ABB RobotStudio station: robotstudio-pick-place.rsstn

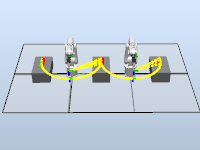
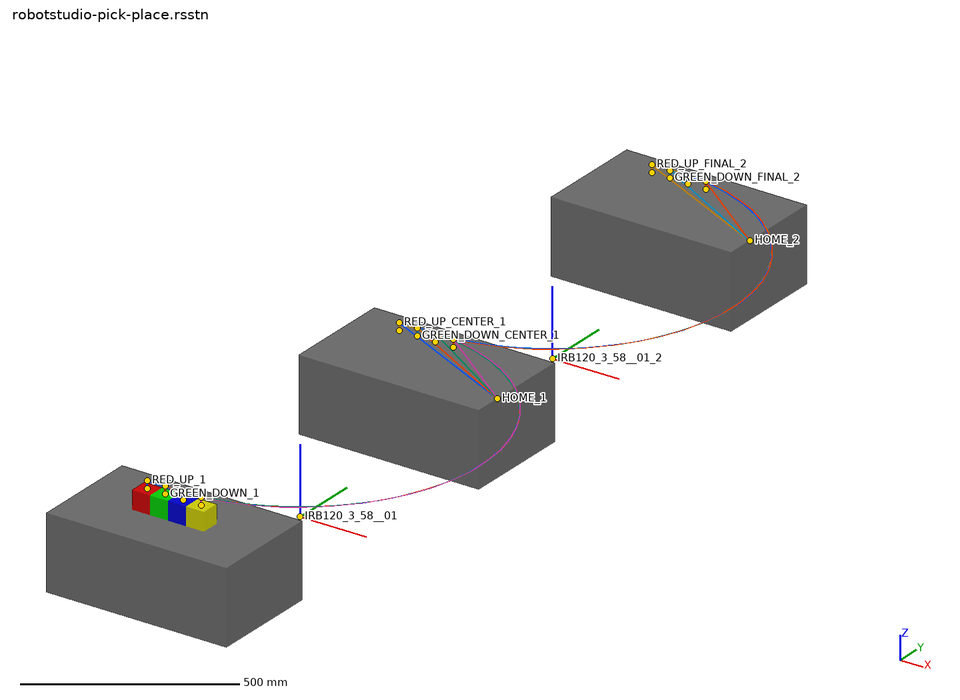
[picture v1: parts stored in the station drawn from their meshes, with robot base, taught points and paths (robot models come from the ABB library and are not in the file)]
Station robotstudio-pick-place (saved by RobotStudio 21.3.9648.0)
Controller PickPlace
  mechanical unit ROB_1: IRB120_3_58__01, 6 joints, base frame (0, 0, 0) mm
  mechanical unit ROB_2: IRB120_3_58__01_2, 6 joints, base frame (0, 1000, 0) mm
Layout (positions relative to the parent item):
  - IRB120_3_58__01 [mechanism, from Robots\IRB120_3_58_G_01.rslib] at (0, 0, 0) mm; joint values [0, 0, 0, 0, 0.5236, 0] (rad or m)
  - IRB120_3_58__01_2 [mechanism, from Robots\IRB120_3_58_G_01.rslib] at (0, 1000, 0) mm; joint values [0, 0, 0, 0, 0.5236, 0] (rad or m)
  - MyTool [mechanism, from Training Objects\myTool.rslib] at (364.35, 0, 594) mm, rotated rx 180 ry 60 rz 180 deg
  - CUBE_1 [part] at (-100, 0, -50) mm, size 50 x 50 x 50 mm
  - CUBE_2 [part] at (-50, 0, -50) mm, size 50 x 50 x 50 mm
  - CUBE_3 [part] at (0, 0, -50) mm, size 50 x 50 x 50 mm
  - CUBE_4 [part] at (50, 0, -50) mm, size 50 x 50 x 50 mm
  - CUBE_1_CENTER [part] at (-100, 1000, -50) mm, size 50 x 50 x 50 mm
  - CUBE_2_CENTER [part] at (-50, 1000, -50) mm, size 50 x 50 x 50 mm
  - CUBE_3_CENTER [part] at (0, 1000, -50) mm, size 50 x 50 x 50 mm
  - CUBE_4_CENTER [part] at (50, 1000, -50) mm, size 50 x 50 x 50 mm
  - CUBE_1_FINAL [part] at (-100, 2000, -50) mm, size 50 x 50 x 50 mm
  - CUBE_2_FINAL [part] at (-50, 2000, -50) mm, size 50 x 50 x 50 mm
  - CUBE_3_FINAL [part] at (0, 2000, -50) mm, size 50 x 50 x 50 mm
  - CUBE_4_FINAL [part] at (50, 2000, -50) mm, size 50 x 50 x 50 mm
  - TABLE_1 [part], size 500 x 300 x 200 mm
  - TABLE_2 [part] at (0, 1000, 0) mm, size 500 x 300 x 200 mm
  - TABLE_3 [part] at (0, 2000, 0) mm, size 500 x 300 x 200 mm
  - MyTool_2 [mechanism, from Training Objects\myTool.rslib] at (364.35, 1000, 594) mm, rotated rx 180 ry 60 rz 180 deg
  - Positioner [smart component, from Components\Positioner.rslib]
      properties: Object=CUBE_1; Position=[0 0 0]; Orientation=[0 0 0]; Reference=Global; ReferenceObject=(none)
  - CollisionSensor [smart component, from Components\CollisionSensor.rslib]
      properties: Object1=MyTool; Object2=CUBE_1; NearMiss=0.01; Part1=(none); Part2=(none); CollisionType=0
  - CollisionSensor_2 [smart component, from Components\CollisionSensor.rslib]
      properties: Object1=MyTool; Object2=CUBE_1_CENTER; NearMiss=0.01; Part1=(none); Part2=(none); CollisionType=0
  - Attacher [smart component, from Components\Attacher.rslib]
      properties: Parent=MyTool; Flange=0; Child=CUBE_1; Mount=false; Offset=[0 0 0]; Orientation=[0 0 0]
  - Detacher [smart component, from Components\Detacher.rslib]
      properties: Child=CUBE_1; KeepPosition=true
  - Positioner_2 [smart component, from Components\Positioner.rslib]
      properties: Object=CUBE_1_CENTER; Position=[0 0 0]; Orientation=[0 0 0]; Reference=Global; ReferenceObject=(none)
  - CollisionSensor_3 [smart component, from Components\CollisionSensor.rslib]
      properties: Object1=MyTool_2; Object2=CUBE_1_CENTER; NearMiss=0.01; Part1=(none); Part2=(none); CollisionType=0
  - CollisionSensor_4 [smart component, from Components\CollisionSensor.rslib]
      properties: Object1=MyTool_2; Object2=CUBE_1_FINAL; NearMiss=0.01; Part1=(none); Part2=(none); CollisionType=0
  - Attacher_2 [smart component, from Components\Attacher.rslib]
      properties: Parent=MyTool_2; Flange=0; Child=CUBE_1; Mount=false; Offset=[0 0 0]; Orientation=[0 0 0]
  - Detacher_2 [smart component, from Components\Detacher.rslib]
      properties: Child=CUBE_1; KeepPosition=true
  - Positioner_3 [smart component, from Components\Positioner.rslib]
      properties: Object=(none); Position=[0 0 0]; Orientation=[0 0 0]; Reference=Global; ReferenceObject=(none)
  - CollisionSensor_5 [smart component, from Components\CollisionSensor.rslib]
      properties: Object1=MyTool; Object2=CUBE_2; NearMiss=0.01; Part1=(none); Part2=(none); CollisionType=0
  - CollisionSensor_6 [smart component, from Components\CollisionSensor.rslib]
      properties: Object1=MyTool; Object2=CUBE_2_CENTER; NearMiss=0.01; Part1=(none); Part2=(none); CollisionType=0
  - Attacher_3 [smart component, from Components\Attacher.rslib]
      properties: Parent=MyTool; Flange=0; Child=CUBE_2; Mount=false; Offset=[0 0 0]; Orientation=[0 0 0]
  - Detacher_3 [smart component, from Components\Detacher.rslib]
      properties: Child=CUBE_2; KeepPosition=true
  - Positioner_4 [smart component, from Components\Positioner.rslib]
      properties: Object=(none); Position=[0 0 0]; Orientation=[0 0 0]; Reference=Global; ReferenceObject=(none)
  - CollisionSensor_7 [smart component, from Components\CollisionSensor.rslib]
      properties: Object1=MyTool_2; Object2=CUBE_2_CENTER; NearMiss=0.01; Part1=(none); Part2=(none); CollisionType=0
  - CollisionSensor_8 [smart component, from Components\CollisionSensor.rslib]
      properties: Object1=MyTool_2; Object2=CUBE_2_FINAL; NearMiss=0.01; Part1=(none); Part2=(none); CollisionType=0
  - Attacher_4 [smart component, from Components\Attacher.rslib]
      properties: Parent=MyTool_2; Flange=0; Child=CUBE_2; Mount=false; Offset=[0 0 0]; Orientation=[0 0 0]
  - Detacher_4 [smart component, from Components\Detacher.rslib]
      properties: Child=CUBE_2; KeepPosition=true
  - Positioner_5 [smart component, from Components\Positioner.rslib]
      properties: Object=(none); Position=[0 0 0]; Orientation=[0 0 0]; Reference=Global; ReferenceObject=(none)
  - CollisionSensor_9 [smart component, from Components\CollisionSensor.rslib]
      properties: Object1=MyTool; Object2=CUBE_3; NearMiss=0.01; Part1=(none); Part2=(none); CollisionType=0
  - CollisionSensor_10 [smart component, from Components\CollisionSensor.rslib]
      properties: Object1=MyTool; Object2=CUBE_3_CENTER; NearMiss=0.01; Part1=(none); Part2=(none); CollisionType=0
  - Attacher_5 [smart component, from Components\Attacher.rslib]
      properties: Parent=MyTool; Flange=0; Child=CUBE_3; Mount=false; Offset=[0 0 0]; Orientation=[0 0 0]
  - Detacher_5 [smart component, from Components\Detacher.rslib]
      properties: Child=CUBE_3; KeepPosition=true
  - Positioner_6 [smart component, from Components\Positioner.rslib]
      properties: Object=(none); Position=[0 0 0]; Orientation=[0 0 0]; Reference=Global; ReferenceObject=(none)
  - CollisionSensor_11 [smart component, from Components\CollisionSensor.rslib]
      properties: Object1=MyTool_2; Object2=CUBE_3; NearMiss=0.01; Part1=(none); Part2=(none); CollisionType=0
  - CollisionSensor_12 [smart component, from Components\CollisionSensor.rslib]
      properties: Object1=MyTool_2; Object2=CUBE_3_FINAL; NearMiss=0.01; Part1=(none); Part2=(none); CollisionType=0
  - Attacher_6 [smart component, from Components\Attacher.rslib]
      properties: Parent=MyTool_2; Flange=0; Child=CUBE_3; Mount=false; Offset=[0 0 0]; Orientation=[0 0 0]
  - Detacher_6 [smart component, from Components\Detacher.rslib]
      properties: Child=CUBE_3; KeepPosition=true
  - Positioner_7 [smart component, from Components\Positioner.rslib]
      properties: Object=(none); Position=[0 0 0]; Orientation=[0 0 0]; Reference=Global; ReferenceObject=(none)
  - CollisionSensor_13 [smart component, from Components\CollisionSensor.rslib]
      properties: Object1=MyTool; Object2=CUBE_4; NearMiss=0.01; Part1=(none); Part2=(none); CollisionType=0
  - CollisionSensor_14 [smart component, from Components\CollisionSensor.rslib]
      properties: Object1=MyTool; Object2=CUBE_4_CENTER; NearMiss=0.01; Part1=(none); Part2=(none); CollisionType=0
  - Attacher_7 [smart component, from Components\Attacher.rslib]
      properties: Parent=MyTool; Flange=0; Child=CUBE_4; Mount=false; Offset=[0 0 0]; Orientation=[0 0 0]
  - Detacher_7 [smart component, from Components\Detacher.rslib]
      properties: Child=CUBE_4; KeepPosition=true
  - Positioner_8 [smart component, from Components\Positioner.rslib]
      properties: Object=CUBE_4_CENTER; Position=[0 0 0]; Orientation=[0 0 0]; Reference=Global; ReferenceObject=(none)
  - CollisionSensor_15 [smart component, from Components\CollisionSensor.rslib]
      properties: Object1=MyTool_2; Object2=CUBE_4_CENTER; NearMiss=0.01; Part1=(none); Part2=(none); CollisionType=0
  - CollisionSensor_16 [smart component, from Components\CollisionSensor.rslib]
      properties: Object1=MyTool_2; Object2=CUBE_4_FINAL; NearMiss=0.01; Part1=(none); Part2=(none); CollisionType=0
  - Attacher_8 [smart component, from Components\Attacher.rslib]
      properties: Parent=MyTool_2; Flange=0; Child=CUBE_4; Mount=false; Offset=[0 0 0]; Orientation=[0 0 0]
  - Detacher_8 [smart component, from Components\Detacher.rslib]
      properties: Child=CUBE_4; KeepPosition=true
Attachment: MyTool is attached to IRB120_3_58__01 / Link6
Attachment: MyTool_2 is attached to IRB120_3_58__01_2 / Link6
Station signals: DI Digital1, DI Digital2, DI Digital3, DI Digital4, DI Digital5, DI Digital6, DI Digital7, DI Digital8
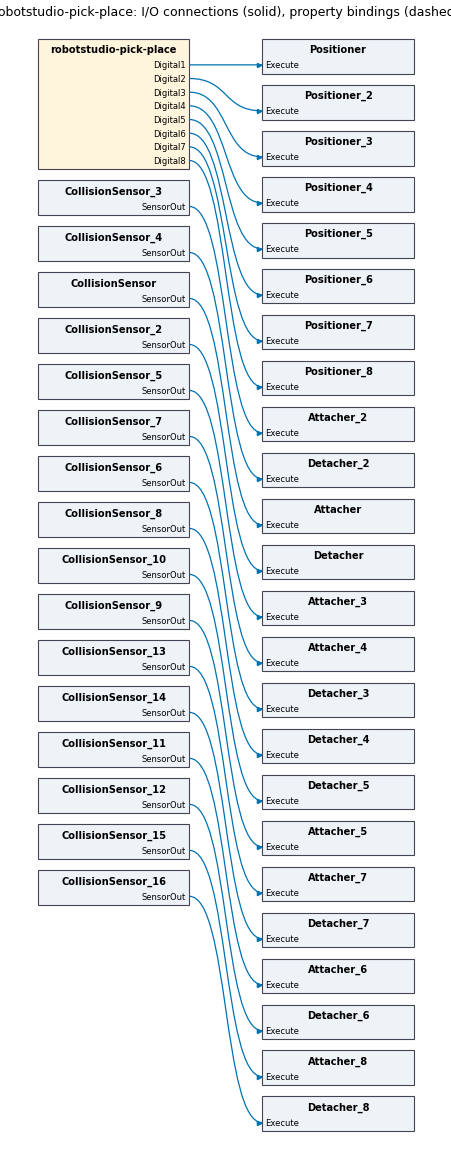
Station logic (signal -> signal, property => property):
  robotstudio-pick-place.Digital1 -> Positioner.Execute
  robotstudio-pick-place.Digital2 -> Positioner_2.Execute
  CollisionSensor_3.SensorOut -> Attacher_2.Execute
  CollisionSensor_4.SensorOut -> Detacher_2.Execute
  CollisionSensor.SensorOut -> Attacher.Execute
  CollisionSensor_2.SensorOut -> Detacher.Execute
  robotstudio-pick-place.Digital3 -> Positioner_3.Execute
  robotstudio-pick-place.Digital4 -> Positioner_4.Execute
  CollisionSensor_5.SensorOut -> Attacher_3.Execute
  CollisionSensor_7.SensorOut -> Attacher_4.Execute
  CollisionSensor_6.SensorOut -> Detacher_3.Execute
  CollisionSensor_8.SensorOut -> Detacher_4.Execute
  robotstudio-pick-place.Digital5 -> Positioner_5.Execute
  CollisionSensor_10.SensorOut -> Detacher_5.Execute
  CollisionSensor_9.SensorOut -> Attacher_5.Execute
  CollisionSensor_13.SensorOut -> Attacher_7.Execute
  CollisionSensor_14.SensorOut -> Detacher_7.Execute
  robotstudio-pick-place.Digital6 -> Positioner_6.Execute
  CollisionSensor_11.SensorOut -> Attacher_6.Execute
  CollisionSensor_12.SensorOut -> Detacher_6.Execute
  robotstudio-pick-place.Digital7 -> Positioner_7.Execute
  CollisionSensor_15.SensorOut -> Attacher_8.Execute
  CollisionSensor_16.SensorOut -> Detacher_8.Execute
  robotstudio-pick-place.Digital8 -> Positioner_8.Execute
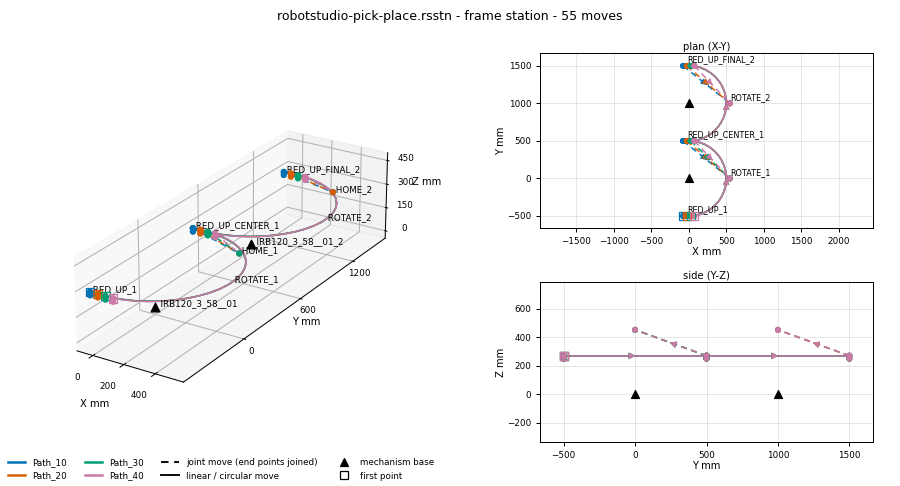
[picture p0: tool path of robotstudio-pick-place.rsstn in frame station, 55 of 55 moves have a stored position in this frame; points joined in program order, loops and branches not executed]
Targets, tools, work objects and paths stored in the station, written as RAPID:
! task T_ROB1
MODULE CalibData
  PERS tooldata MyTool:=[TRUE,[[31.792631019,0,229.638935148],[0.945518576,0,0.325568154,0]],[1,[0,0,1],[1,0,0,0],0,0,0]];
ENDMODULE

! task T_ROB1
MODULE Module1
  CONST robtarget RED_DOWN_1:=[[-75,-500,250],[0,0.707106781,0.707106781,0],[-2,0,-1,0],[9E+09,9E+09,9E+09,9E+09,9E+09,9E+09]];
  CONST robtarget RED_UP_1:=[[-75,-500,270],[0,0.707106781,0.707106781,0],[-2,0,-1,0],[9E+09,9E+09,9E+09,9E+09,9E+09,9E+09]];
  CONST robtarget RED_DOWN_CENTER_1:=[[-75,500,250],[0,-0.707106781,0.707106781,0],[0,0,0,0],[9E+09,9E+09,9E+09,9E+09,9E+09,9E+09]];
  CONST robtarget RED_UP_CENTER_1:=[[-75,500,270],[0,-0.707106781,0.707106781,0],[0,0,0,0],[9E+09,9E+09,9E+09,9E+09,9E+09,9E+09]];
  CONST robtarget ROTATE_1:=[[500,0,270],[0,0,1,0],[0,0,0,0],[9E+09,9E+09,9E+09,9E+09,9E+09,9E+09]];
  CONST robtarget HOME_1:=[[547.330665099,0,451.64730631],[0.190808996,0,0.981627183,0],[0,0,0,0],[9E+09,9E+09,9E+09,9E+09,9E+09,9E+09]];
  CONST robtarget GREEN_DOWN_1:=[[-25,-500,250],[0,0.707106781,0.707106781,0],[0,0,0,0],[9E+09,9E+09,9E+09,9E+09,9E+09,9E+09]];
  CONST robtarget GREEN_UP_1:=[[-25,-500,270],[0,0.707106781,0.707106781,0],[0,0,0,0],[9E+09,9E+09,9E+09,9E+09,9E+09,9E+09]];
  CONST robtarget GREEN_DOWN_CENTER_1:=[[-25,500,250],[0,-0.707106781,0.707106781,0],[0,0,0,0],[9E+09,9E+09,9E+09,9E+09,9E+09,9E+09]];
  CONST robtarget GREEN_UP_CENTER_1:=[[-25,500,270],[0,-0.707106781,0.707106781,0],[0,0,0,0],[9E+09,9E+09,9E+09,9E+09,9E+09,9E+09]];
  CONST robtarget BLUE_DOWN_1:=[[25,-500,250],[0,0.707106781,0.707106781,0],[-1,-1,0,0],[9E+09,9E+09,9E+09,9E+09,9E+09,9E+09]];
  CONST robtarget BLUE_UP_1:=[[25,-500,270],[0,0.707106781,0.707106781,0],[0,0,0,0],[9E+09,9E+09,9E+09,9E+09,9E+09,9E+09]];
  CONST robtarget BLUE_DOWN_CENTER_1:=[[25,500,250],[0,-0.707106781,0.707106781,0],[0,0,-1,0],[9E+09,9E+09,9E+09,9E+09,9E+09,9E+09]];
  CONST robtarget BLUE_UP_CENTER_1:=[[25,500,270],[0,-0.707106781,0.707106781,0],[0,0,-1,0],[9E+09,9E+09,9E+09,9E+09,9E+09,9E+09]];
  CONST robtarget YELLOW_DOWN_1:=[[75,-500,250],[0,0.707106781,0.707106781,0],[-1,-1,0,0],[9E+09,9E+09,9E+09,9E+09,9E+09,9E+09]];
  CONST robtarget YELLOW_UP_1:=[[75,-500,270],[0,0.707106781,0.707106781,0],[0,0,0,0],[9E+09,9E+09,9E+09,9E+09,9E+09,9E+09]];
  CONST robtarget YELLOW_DOWN_CENTER_1:=[[75,500,250],[0,-0.707106781,0.707106781,0],[0,0,-1,0],[9E+09,9E+09,9E+09,9E+09,9E+09,9E+09]];
  CONST robtarget YELLOW_UP_CENTER_1:=[[75,500,270],[0,-0.707106781,0.707106781,0],[0,0,-1,0],[9E+09,9E+09,9E+09,9E+09,9E+09,9E+09]];
  PROC Path_10()
    MoveJ RED_UP_1,v1000,fine,MyTool\WObj:=wobj0;
    MoveL RED_DOWN_1,v1000,fine,MyTool\WObj:=wobj0;
    MoveL RED_UP_1,v1000,z100,MyTool\WObj:=wobj0;
    MoveC ROTATE_1,RED_UP_CENTER_1,v1000,z100,MyTool\WObj:=wobj0;
    MoveL RED_DOWN_CENTER_1,v1000,z100,MyTool\WObj:=wobj0;
    MoveL RED_UP_CENTER_1,v1000,z100,MyTool\WObj:=wobj0;
    MoveJ HOME_1,v1000,fine,MyTool\WObj:=wobj0;
  ENDPROC
  PROC Path_20()
    MoveJ GREEN_UP_1,v1000,fine,MyTool\WObj:=wobj0;
    MoveL GREEN_DOWN_1,v1000,z100,MyTool\WObj:=wobj0;
    MoveL GREEN_UP_1,v1000,z100,MyTool\WObj:=wobj0;
    MoveC ROTATE_1,GREEN_UP_CENTER_1,v1000,z100,MyTool\WObj:=wobj0;
    MoveL GREEN_DOWN_CENTER_1,v1000,z100,MyTool\WObj:=wobj0;
    MoveL GREEN_UP_CENTER_1,v1000,z100,MyTool\WObj:=wobj0;
    MoveJ HOME_1,v1000,fine,MyTool\WObj:=wobj0;
  ENDPROC
  PROC Path_30()
    MoveJ BLUE_UP_1,v1000,fine,MyTool\WObj:=wobj0;
    MoveL BLUE_DOWN_1,v1000,z100,MyTool\WObj:=wobj0;
    MoveL BLUE_UP_1,v1000,z100,MyTool\WObj:=wobj0;
    MoveC ROTATE_1,BLUE_UP_CENTER_1,v1000,z100,MyTool\WObj:=wobj0;
    MoveL BLUE_DOWN_CENTER_1,v1000,z100,MyTool\WObj:=wobj0;
    MoveL BLUE_UP_CENTER_1,v1000,z100,MyTool\WObj:=wobj0;
    MoveJ HOME_1,v1000,fine,MyTool\WObj:=wobj0;
  ENDPROC
  PROC Path_40()
    MoveJ YELLOW_UP_1,v1000,fine,MyTool\WObj:=wobj0;
    MoveL YELLOW_DOWN_1,v1000,z100,MyTool\WObj:=wobj0;
    MoveL YELLOW_UP_1,v1000,z100,MyTool\WObj:=wobj0;
    MoveC ROTATE_1,YELLOW_UP_CENTER_1,v1000,z100,MyTool\WObj:=wobj0;
    MoveL YELLOW_DOWN_CENTER_1,v1000,z100,MyTool\WObj:=wobj0;
    MoveL YELLOW_UP_CENTER_1,v1000,z100,MyTool\WObj:=wobj0;
    MoveJ HOME_1,v1000,fine,MyTool\WObj:=wobj0;
  ENDPROC
ENDMODULE

! task T_ROB2
MODULE CalibData
  PERS tooldata MyTool:=[TRUE,[[31.792631019,0,229.638935148],[0.945518576,0,0.325568154,0]],[1,[0,0,1],[1,0,0,0],0,0,0]];
ENDMODULE

! task T_ROB2
MODULE Module1
  CONST robtarget RED_DOWN_2:=[[-75,500,250],[0,0.707106781,0.707106781,0],[-2,0,-1,0],[9E+09,9E+09,9E+09,9E+09,9E+09,9E+09]];
  CONST robtarget RED_UP_2:=[[-75,500,270],[0,0.707106781,0.707106781,0],[-2,0,-1,0],[9E+09,9E+09,9E+09,9E+09,9E+09,9E+09]];
  CONST robtarget RED_DOWN_FINAL_2:=[[-75,1500,250],[0,-0.707106781,0.707106781,0],[1,-1,0,0],[9E+09,9E+09,9E+09,9E+09,9E+09,9E+09]];
  CONST robtarget RED_UP_FINAL_2:=[[-75,1500,270],[0,-0.707106781,0.707106781,0],[1,-1,0,0],[9E+09,9E+09,9E+09,9E+09,9E+09,9E+09]];
  CONST robtarget ROTATE_2:=[[500,1000,270],[0,0,1,0],[0,0,0,0],[9E+09,9E+09,9E+09,9E+09,9E+09,9E+09]];
  CONST robtarget HOME_2:=[[547.330665099,1000,451.64730631],[0.190808996,0,0.981627183,0],[0,0,0,0],[9E+09,9E+09,9E+09,9E+09,9E+09,9E+09]];
  CONST robtarget GREEN_DOWN_2:=[[-25,500,250],[0,0.707106781,0.707106781,0],[-2,0,-1,0],[9E+09,9E+09,9E+09,9E+09,9E+09,9E+09]];
  CONST robtarget GREEN_UP_2:=[[-25,500,270],[0,0.707106781,0.707106781,0],[-2,0,-1,0],[9E+09,9E+09,9E+09,9E+09,9E+09,9E+09]];
  CONST robtarget GREEN_DOWN_FINAL_2:=[[-25,1500,250],[0,-0.707106781,0.707106781,0],[1,-1,0,0],[9E+09,9E+09,9E+09,9E+09,9E+09,9E+09]];
  CONST robtarget GREEN_UP_FINAL_2:=[[-25,1500,270],[0,-0.707106781,0.707106781,0],[1,-1,0,0],[9E+09,9E+09,9E+09,9E+09,9E+09,9E+09]];
  CONST robtarget BLUE_DOWN_2:=[[25,500,250],[0,0.707106781,0.707106781,0],[-1,-1,0,0],[9E+09,9E+09,9E+09,9E+09,9E+09,9E+09]];
  CONST robtarget BLUE_UP_2:=[[25,500,270],[0,0.707106781,0.707106781,0],[0,0,0,0],[9E+09,9E+09,9E+09,9E+09,9E+09,9E+09]];
  CONST robtarget BLUE_DOWN_FINAL_2:=[[25,1500,250],[0,-0.707106781,0.707106781,0],[0,0,-1,0],[9E+09,9E+09,9E+09,9E+09,9E+09,9E+09]];
  CONST robtarget BLUE_UP_FINAL_2:=[[25,1500,270],[0,-0.707106781,0.707106781,0],[0,0,-1,0],[9E+09,9E+09,9E+09,9E+09,9E+09,9E+09]];
  CONST robtarget YELLOW_DOWN_2:=[[75,500,250],[0,0.707106781,0.707106781,0],[-1,-1,0,0],[9E+09,9E+09,9E+09,9E+09,9E+09,9E+09]];
  CONST robtarget YELLOW_UP_2:=[[75,500,270],[0,0.707106781,0.707106781,0],[0,0,0,0],[9E+09,9E+09,9E+09,9E+09,9E+09,9E+09]];
  CONST robtarget YELLOW_DOWN_FINAL_2:=[[75,1500,250],[0,-0.707106781,0.707106781,0],[0,0,-1,0],[9E+09,9E+09,9E+09,9E+09,9E+09,9E+09]];
  CONST robtarget YELLOW_UP_FINAL_2:=[[75,1500,270],[0,-0.707106781,0.707106781,0],[0,0,-1,0],[9E+09,9E+09,9E+09,9E+09,9E+09,9E+09]];
  PROC Path_10()
    MoveJ RED_UP_2,v1000,fine,MyTool\WObj:=wobj0;
    MoveL RED_DOWN_2,v1000,z100,MyTool\WObj:=wobj0;
    MoveL RED_UP_2,v1000,z100,MyTool\WObj:=wobj0;
    MoveC ROTATE_2,RED_UP_FINAL_2,v1000,z100,MyTool\WObj:=wobj0;
    MoveL RED_DOWN_FINAL_2,v1000,z100,MyTool\WObj:=wobj0;
    MoveL RED_UP_FINAL_2,v1000,z100,MyTool\WObj:=wobj0;
    MoveJ HOME_2,v1000,fine,MyTool\WObj:=wobj0;
  ENDPROC
  PROC Path_20()
    MoveJ GREEN_UP_2,v1000,fine,MyTool\WObj:=wobj0;
    MoveL GREEN_DOWN_2,v1000,z100,MyTool\WObj:=wobj0;
    MoveL GREEN_UP_2,v1000,z100,MyTool\WObj:=wobj0;
    MoveC ROTATE_2,GREEN_UP_FINAL_2,v1000,z100,MyTool\WObj:=wobj0;
    MoveL GREEN_DOWN_FINAL_2,v1000,z100,MyTool\WObj:=wobj0;
    MoveL GREEN_UP_FINAL_2,v1000,z100,MyTool\WObj:=wobj0;
    MoveJ HOME_2,v1000,fine,MyTool\WObj:=wobj0;
  ENDPROC
  PROC Path_30()
    MoveJ BLUE_UP_2,v1000,fine,MyTool\WObj:=wobj0;
    MoveL BLUE_DOWN_2,v1000,z100,MyTool\WObj:=wobj0;
    MoveL BLUE_UP_2,v1000,z100,MyTool\WObj:=wobj0;
    MoveC ROTATE_2,BLUE_UP_FINAL_2,v1000,z100,MyTool\WObj:=wobj0;
    MoveL BLUE_DOWN_FINAL_2,v1000,z100,MyTool\WObj:=wobj0;
    MoveJ BLUE_UP_FINAL_2,v1000,fine,MyTool\WObj:=wobj0;
  ENDPROC
  PROC Path_40()
    MoveJ YELLOW_UP_2,v1000,fine,MyTool\WObj:=wobj0;
    MoveL YELLOW_DOWN_2,v1000,z100,MyTool\WObj:=wobj0;
    MoveL YELLOW_UP_2,v1000,z100,MyTool\WObj:=wobj0;
    MoveC ROTATE_2,YELLOW_UP_FINAL_2,v1000,z100,MyTool\WObj:=wobj0;
    MoveL YELLOW_DOWN_FINAL_2,v1000,z100,MyTool\WObj:=wobj0;
    MoveL YELLOW_UP_FINAL_2,v1000,z100,MyTool\WObj:=wobj0;
    MoveJ HOME_2,v1000,fine,MyTool\WObj:=wobj0;
  ENDPROC
ENDMODULE

